///EL1252 | XFC, 2-channel digital input terminal with time stamp
FUNCTION_BLOCK EL1252

VAR_INPUT
	En: BOOL;
	iTerminal_ID : INT;
	ErrorSystem : POINTER TO ST_ErrorSystem;
END_VAR

VAR_OUTPUT
	EnO: BOOL;
	bDi_1: BOOL;
	bDi_2: BOOL;
	nDcTimeOnLatchPos_1: ULINT;
	nDcTimeOnLatchNeg_1: ULINT;
	nDcTimeOnLatchPos_2: ULINT;
	nDcTimeOnLatchNeg_2: ULINT;
	bError: BOOL;
END_VAR

VAR
	Channel_1_Input AT %I*: BOOL;
	Channel_2_Input AT %I*: BOOL;
	Latch_LatchPos1 AT %I*: ULINT;
	Latch_LatchNeg1 AT %I*: ULINT;
	Latch_LatchPos2 AT %I*: ULINT;
	Latch_LatchNeg2 AT %I*: ULINT;
	WcState_WcState AT %I*: BOOL;
	InfoData_State AT %I*: UINT;
	
	//FB-s
	fbTerminalError : FB_TerminalError;
END_VAR

(*
*	No Error System related registers other than WcState and InfoData_State
*)

EnO:=En;

//Error FB instance
fbTerminalError(
	En := TRUE,
	iTerminal_ID := iTerminal_ID,
	bWcState := WcState_WcState,
	uiInfoData_State := InfoData_State,
	pErrorSystem := ErrorSystem,
	bError => bError,
);

IF En THEN
	IF bError=FALSE THEN
		bDi_1:=Channel_1_Input;
		bDi_2:=Channel_2_Input;
		nDcTimeOnLatchPos_1:=Latch_LatchPos1;
		nDcTimeOnLatchNeg_1:=Latch_LatchNeg1;
		nDcTimeOnLatchPos_2:=Latch_LatchPos2;
		nDcTimeOnLatchNeg_2:=Latch_LatchNeg2;
	ELSE
		bDi_1:=FALSE;
		bDi_2:=FALSE;
		nDcTimeOnLatchPos_1:=0;
		nDcTimeOnLatchNeg_1:=0;
		nDcTimeOnLatchPos_2:=0;
		nDcTimeOnLatchNeg_2:=0;
	END_IF
END_IF

END_FUNCTION_BLOCK

(* stored: Version 1.1.0.1, ProductVersion 3.1.4022.10
   POU EL1252: Id {9414ba14-6645-4599-8459-3b12adb78306}, SpecialFunc None *)
